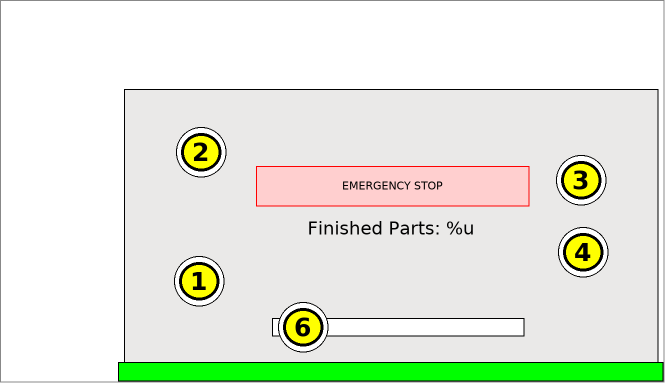
VISUALIZATION TableState  // 665x383
    Rectangle (124,89 534x279), "Finished Parts: %u", text variable: MAIN.FinishedParts, colour toggle: NOT MAIN.MasterRunStop
    Ellipse (176,127 50x50), "2"
    Ellipse (174,256 50x50), "1"
    Ellipse (556,155 50x50), "3"
    Ellipse (558,227 50x50), "4"
    Rectangle (272,318 252x18)
    Ellipse (278,302 50x50), "6"
    Ellipse (181,133 40x38), "2", colour toggle: MAIN.Station_2_Timer.Q, invisible if: NOT MAIN.station_2_sensor
    Ellipse (179,262 40x38), "1", colour toggle: MAIN.Station_1_Timer.Q, invisible if: NOT MAIN.station_1_sensor
    Ellipse (561,161 40x38), "3", colour toggle: MAIN.Station_3_Timer.Q, invisible if: NOT MAIN.station_3_sensor
    Ellipse (563,233 40x38), "4", colour toggle: MAIN.Station_4_Timer.Q, invisible if: NOT MAIN.station_4_sensor
    Ellipse (283,308 40x38), "6", colour toggle: MAIN.station_6_sensor, invisible if: NOT MAIN.station_6_sensor
    Rectangle (118,362 545x19), colour toggle: NOT MAIN.LightCurtainStatus
    Rectangle (256,166 273x40), "EMERGENCY STOP", invisible if: MAIN.EStopButtonStatus
END_VISUALIZATION

(* stored: Version 1.1.0.1, ProductVersion 3.1.0.36
   Visu TableState: Id {01e48f87-6a50-4fdf-8ab2-d75ef98a4604} *)
